PROGRAM MAIN
VAR
END_VAR

END_PROGRAM

(* stored: Version 1.1.0.1
   POU MAIN: Id {cd5ed0b3-00ae-44ee-b916-3c7c72288cdf} *)
